(* IEC 61131-3 sources: ml2plc/benchmarks/st, 42 files *)

(* ---- CNN1.st ---- *)
FUNCTION_BLOCK CNN1_FB

    (* Model Inputs/Outputs *)
VAR_INPUT
    input_data : REAL;
END_VAR

VAR_OUTPUT
    output_data : ARRAY[0..2] OF REAL;
END_VAR

VAR CONSTANT
    weights_0 : ARRAY[0..5] OF REAL := [-0.757294893, 1.60322511, -0.810065687, -0.0401188135, -0.0341094136, 2.28848505];
    bias_0 : ARRAY[0..5] OF REAL := [0, -0.327996045, 0, 0, 0, -0.425784826];

    weights_2 : ARRAY[0..95] OF REAL := [0.387440026, -0.331604958, -0.485271782, -0.178175241, -0.261189312, -0.126141995, -0.41867274, 0.10701102, -0.504957795, -0.0640092492, -0.506339848, -0.0112774968, -0.248149365, 0.370121658, 0.102361083, 0.514361918, 2.27920318, -2.03401303, 2.57838869, 0.345396936, 1.7697078, 2.31489539, 1.82641065, 0.116435051, 2.60688972, -0.141314536, 0.0899649858, -0.115778536, -0.130346328, -2.0967865, 1.73134959, 1.73764074, -0.125548214, -0.418661654, 0.42383492, 0.245940804, -0.231652409, -0.521428883, -0.369046271, 0.500959337, 0.39457792, -0.498766184, 0.505615175, 0.00158774853, -0.358177781, 0.0681350231, 0.211269855, 0.317975223, 0.470600903, -0.22380206, -0.221884102, 0.369123101, -0.365577281, 0.470880032, 0.0877029896, -0.22456941, 0.125117779, 0.0604217052, 0.403043449, 0.0515841246, 0.360347748, 0.176390409, 0.499794424, 0.4554739, 0.357078254, -0.20554477, -0.338528842, -0.346329391, -0.316419125, -0.192169428, 0.340339243, -0.170743108, 0.503388941, 0.431303263, 0.182139158, 0.344671071, 0.0957750082, -0.455443144, 0.516620576, -0.12648204, 2.20542169, -1.42068136, 1.77867258, -0.279205918, 1.31937492, 2.40089417, 1.49984801, -0.381873012, 2.37344623, -0.157825798, -0.164687812, -0.438219547, -0.030656606, -0.809033334, 1.04967833, 1.52932751];
    bias_2 : ARRAY[0..15] OF REAL := [-0.00126687379, 1.46715438, -0.0669283643, 0, -0.544165969, -0.00420819549, -0.593534648, 0, -0.00139115693, 0, 0, 0, 0, 1.40235019, -0.471719682, -0.589310586];

    weights_3 : ARRAY[0..47] OF REAL := [-2.44326067, 1.56872427, 1.00637841, 2.21994734, -0.0721509904, -2.70681095, -2.57062817, 0.8563025, 1.35775805, 0.436492383, -0.214310527, 0.435115576, -0.357676566, -2.57688642, 2.20074344, -1.96935773, 1.55129766, 1.27391887, -0.475576401, -2.55197287, 1.79706705, -0.406806469, -0.373194754, 0.021515131, -1.98918331, 1.86888134, 1.35972965, 0.224319875, -0.156571329, -0.38576901, -0.264996111, -0.172905713, 0.307211518, 0.210194111, -0.266009122, -0.164967567, -0.275477469, 0.512401879, 0.539515197, 1.5903399, -0.0624566786, -2.02082109, -1.80255735, -3.25323439, 2.98463917, -0.251099586, -2.6509831, 1.72883391];
    bias_3 : ARRAY[0..2] OF REAL := [0.74891752, -0.036865145, -0.95004487];

END_VAR

VAR
    (* Merged variables from all regions *)
    buffer_0 : ARRAY[0..5] OF REAL;
    buffer_1 : ARRAY[0..15] OF REAL;

    (* Temporary computation variables *)
    i : DINT;
    j : DINT;
    t : DINT;
    sum : REAL;
    (* Computation helpers *)
    max_val : REAL;
    exp_val : REAL;
    exp_sum : REAL;
    (* Spatial loop variables *)
    oc : DINT;
    oh : DINT;
    ow : DINT;
    ic : DINT;
    kh : DINT;
    kw : DINT;
    ih : DINT;
    iw : DINT;
END_VAR

(* Forward pass execution *)

(* Region: r0 [ACYCLIC] *)
(* Acyclic Region r0 *)
(* Layer 0: Conv2D  in=1x1x1  out=6x1x1  kernel=1x1  stride=1x1  pad=(0, 0, 0, 0)  group=1 *)
FOR oc := 0 TO 5 DO
    FOR oh := 0 TO 0 DO
        FOR ow := 0 TO 0 DO
            sum := bias_0[oc];
            FOR ic := 0 TO 0 DO
                FOR kh := 0 TO 0 DO
                    FOR kw := 0 TO 0 DO
                        ih := oh * 1 - 0 + kh;
                        iw := ow * 1 - 0 + kw;
                        sum := sum + input_data * weights_0[oc * 1 + ic * 1 + kh * 1 + kw];
                    END_FOR;
                END_FOR;
            END_FOR;
            buffer_1[oc * 1 + oh * 1 + ow] := sum;
        END_FOR;
    END_FOR;
END_FOR;

(* Layer 1: Activation (RELU) *)
FOR i := 0 TO 5 DO
    buffer_0[i] := MAX(buffer_1[i], 0.0);
END_FOR;

(* Layer 2: Fused Linear + RELU *)
FOR j := 0 TO 15 DO
    sum := 0.0;
    FOR i := 0 TO 5 DO
        sum := sum + buffer_0[i] * weights_2[i * 16 + j];
    END_FOR;
buffer_1[j] := MAX(sum + bias_2[j], 0.0);
END_FOR;

(* Layer 3: Fused Linear + SOFTMAX *)
FOR j := 0 TO 2 DO
    sum := 0.0;
    FOR i := 0 TO 15 DO
        sum := sum + buffer_1[i] * weights_3[i * 3 + j];
    END_FOR;
output_data[j] := sum + bias_3[j];
END_FOR;

(* Softmax: find max *)
max_val := output_data[0];
FOR i := 1 TO 2 DO
    IF output_data[i] > max_val THEN
        max_val := output_data[i];
    END_IF;
END_FOR;

(* Softmax: compute exponentials and sum *)
exp_sum := 0.0;
FOR i := 0 TO 2 DO
    output_data[i] := EXP(output_data[i] - max_val);
    exp_sum := exp_sum + output_data[i];
END_FOR;

(* Softmax: normalize *)
FOR i := 0 TO 2 DO
    output_data[i] := output_data[i] / exp_sum;
END_FOR;

END_FUNCTION_BLOCK

(* ---- CNN1_straton.st ---- *)
FUNCTION_BLOCK CNN1_FB

    (* Model Inputs/Outputs *)
VAR_INPUT
    input_data : REAL;
END_VAR

VAR_OUTPUT
    output_data : ARRAY[0..2] OF REAL;
END_VAR

VAR
    CONSTANT weights_0 : ARRAY[0..5] OF REAL := [-0.757294893, 1.60322511, -0.810065687, -0.0401188135, -0.0341094136, 2.28848505];
    CONSTANT bias_0 : ARRAY[0..5] OF REAL := [0, -0.327996045, 0, 0, 0, -0.425784826];
    CONSTANT weights_2 : ARRAY[0..95] OF REAL := [0.387440026, -0.331604958, -0.485271782, -0.178175241, -0.261189312, -0.126141995, -0.41867274, 0.10701102, -0.504957795, -0.0640092492, -0.506339848, -0.0112774968, -0.248149365, 0.370121658, 0.102361083, 0.514361918, 2.27920318, -2.03401303, 2.57838869, 0.345396936, 1.7697078, 2.31489539, 1.82641065, 0.116435051, 2.60688972, -0.141314536, 0.0899649858, -0.115778536, -0.130346328, -2.0967865, 1.73134959, 1.73764074, -0.125548214, -0.418661654, 0.42383492, 0.245940804, -0.231652409, -0.521428883, -0.369046271, 0.500959337, 0.39457792, -0.498766184, 0.505615175, 0.00158774853, -0.358177781, 0.0681350231, 0.211269855, 0.317975223, 0.470600903, -0.22380206, -0.221884102, 0.369123101, -0.365577281, 0.470880032, 0.0877029896, -0.22456941, 0.125117779, 0.0604217052, 0.403043449, 0.0515841246, 0.360347748, 0.176390409, 0.499794424, 0.4554739, 0.357078254, -0.20554477, -0.338528842, -0.346329391, -0.316419125, -0.192169428, 0.340339243, -0.170743108, 0.503388941, 0.431303263, 0.182139158, 0.344671071, 0.0957750082, -0.455443144, 0.516620576, -0.12648204, 2.20542169, -1.42068136, 1.77867258, -0.279205918, 1.31937492, 2.40089417, 1.49984801, -0.381873012, 2.37344623, -0.157825798, -0.164687812, -0.438219547, -0.030656606, -0.809033334, 1.04967833, 1.52932751];
    CONSTANT bias_2 : ARRAY[0..15] OF REAL := [-0.00126687379, 1.46715438, -0.0669283643, 0, -0.544165969, -0.00420819549, -0.593534648, 0, -0.00139115693, 0, 0, 0, 0, 1.40235019, -0.471719682, -0.589310586];
    CONSTANT weights_3 : ARRAY[0..47] OF REAL := [-2.44326067, 1.56872427, 1.00637841, 2.21994734, -0.0721509904, -2.70681095, -2.57062817, 0.8563025, 1.35775805, 0.436492383, -0.214310527, 0.435115576, -0.357676566, -2.57688642, 2.20074344, -1.96935773, 1.55129766, 1.27391887, -0.475576401, -2.55197287, 1.79706705, -0.406806469, -0.373194754, 0.021515131, -1.98918331, 1.86888134, 1.35972965, 0.224319875, -0.156571329, -0.38576901, -0.264996111, -0.172905713, 0.307211518, 0.210194111, -0.266009122, -0.164967567, -0.275477469, 0.512401879, 0.539515197, 1.5903399, -0.0624566786, -2.02082109, -1.80255735, -3.25323439, 2.98463917, -0.251099586, -2.6509831, 1.72883391];
    CONSTANT bias_3 : ARRAY[0..2] OF REAL := [0.74891752, -0.036865145, -0.95004487];
END_VAR

VAR
    (* Merged variables from all regions *)
    buffer_0 : ARRAY[0..5] OF REAL;
    buffer_1 : ARRAY[0..15] OF REAL;

    (* Temporary computation variables *)
    i : DINT;
    j : DINT;
    t : DINT;
    sum : REAL;
    (* Computation helpers *)
    max_val : REAL;
    exp_val : REAL;
    exp_sum : REAL;
    (* Spatial loop variables *)
    oc : DINT;
    oh : DINT;
    ow : DINT;
    ic : DINT;
    kh : DINT;
    kw : DINT;
    ih : DINT;
    iw : DINT;
END_VAR

(* Forward pass execution *)

(* Region: r0 [ACYCLIC] *)
(* Acyclic Region r0 *)
(* Layer 0: Conv2D  in=1x1x1  out=6x1x1  kernel=1x1  stride=1x1  pad=(0, 0, 0, 0)  group=1 *)
FOR oc := 0 TO 5 DO
    FOR oh := 0 TO 0 DO
        FOR ow := 0 TO 0 DO
            sum := bias_0[oc];
            FOR ic := 0 TO 0 DO
                FOR kh := 0 TO 0 DO
                    FOR kw := 0 TO 0 DO
                        ih := oh * 1 - 0 + kh;
                        iw := ow * 1 - 0 + kw;
                        sum := sum + input_data * weights_0[oc * 1 + ic * 1 + kh * 1 + kw];
                    END_FOR;
                END_FOR;
            END_FOR;
            buffer_1[oc * 1 + oh * 1 + ow] := sum;
        END_FOR;
    END_FOR;
END_FOR;

(* Layer 1: Activation (RELU) *)
FOR i := 0 TO 5 DO
    buffer_0[i] := MAX(buffer_1[i], 0.0);
END_FOR;

(* Layer 2: Fused Linear + RELU *)
FOR j := 0 TO 15 DO
    sum := 0.0;
    FOR i := 0 TO 5 DO
        sum := sum + buffer_0[i] * weights_2[i * 16 + j];
    END_FOR;
buffer_1[j] := MAX(sum + bias_2[j], 0.0);
END_FOR;

(* Layer 3: Fused Linear + SOFTMAX *)
FOR j := 0 TO 2 DO
    sum := 0.0;
    FOR i := 0 TO 15 DO
        sum := sum + buffer_1[i] * weights_3[i * 3 + j];
    END_FOR;
output_data[j] := sum + bias_3[j];
END_FOR;

(* Softmax: find max *)
max_val := output_data[0];
FOR i := 1 TO 2 DO
    IF output_data[i] > max_val THEN
        max_val := output_data[i];
    END_IF;
END_FOR;

(* Softmax: compute exponentials and sum *)
exp_sum := 0.0;
FOR i := 0 TO 2 DO
    output_data[i] := EXP(output_data[i] - max_val);
    exp_sum := exp_sum + output_data[i];
END_FOR;

(* Softmax: normalize *)
FOR i := 0 TO 2 DO
    output_data[i] := output_data[i] / exp_sum;
END_FOR;

END_FUNCTION_BLOCK

(* ---- CNN2.st ---- *)
FUNCTION_BLOCK CNN2_FB

    (* Model Inputs/Outputs *)
VAR_INPUT
    input_data : REAL;
END_VAR

VAR_OUTPUT
    output_data : ARRAY[0..2] OF REAL;
END_VAR

VAR CONSTANT
    weights_0 : ARRAY[0..9] OF REAL := [-0.262705386, 0.779935002, 1.03506529, 0.632895529, -0.312737316, -0.310815006, 1.04849136, 0.870586991, -0.33241713, 0.675958574];
    bias_0 : ARRAY[0..9] OF REAL := [0, -0.171853036, 0.155731231, -0.141236976, 0, 0.388507366, -0.176535189, -0.0690641031, 0, -0.149513766];

    weights_2 : ARRAY[0..99] OF REAL := [-0.0687341988, -0.505324185, -0.171715677, -0.380084217, 0.443206012, -0.165993631, -0.00731980801, -0.294861794, -0.329322875, -0.340971529, -0.39975965, -1.21721697, 0.0680034459, -1.40909934, 0.224685371, 0.851948142, -0.889827847, -0.095493108, -0.157179385, -1.28536439, -0.545177042, -1.34768605, 0.0538454317, -0.994832158, 0.527012348, 0.700168669, -1.15851235, -0.457079113, -0.00149732828, -0.467484027, 0.178472638, -1.06804824, 0.428462833, -0.918258965, -0.139204293, 0.417420805, -0.467564315, 0.0089803664, -0.24426356, -1.38583362, -0.463089764, 0.807691395, 0.923243821, 0.796885252, 0.0120127201, -0.49810043, 0.873528719, 0.914482772, 0.53928721, 0.734467626, 0.278324604, 1.19621909, 0.403788477, 1.62108636, 0.500351071, -0.523164451, 0.972507596, 0.644115269, -0.138118327, 1.47070789, 0.209766984, 0.853332102, 0.699123144, 0.846534193, 0.213573575, 0.678547621, 1.08085775, 0.551357388, 0.0911467671, 0.56043458, 0.102282166, 0.877178192, 1.12506092, 0.902248561, 0.383322537, 0.205958784, 1.27946091, 0.450389624, 0.0967945457, 1.4164356, -0.126412362, 0.519436717, -0.367547452, -0.315561593, 0.464017153, -0.335243285, -0.132026047, 0.0108332634, -0.113086581, 0.499188185, -0.124567181, 0.982846677, 0.764017642, 0.814776838, 0.0450161695, -0.607075572, 1.12853694, 1.060583, -0.528354645, 1.37106454];
    bias_2 : ARRAY[0..9] OF REAL := [0, 0.411672026, 0.443880588, 0.573848665, -0.0798636526, -0.125108838, 0.121025026, 0.385259449, 0, -0.19617413];

    weights_4 : ARRAY[0..159] OF REAL := [-0.201477349, 0.413015246, 0.0206950307, -0.0461762249, 0.247961462, -0.0568501949, 0.0383369327, -0.259854972, -0.444527179, 0.354037642, -0.150492162, -0.45852077, -0.0717066824, 0.0723364949, -0.436497748, 0.205825031, -0.853246808, -0.203027666, 1.20550728, -0.617461145, -0.294606566, -0.758126974, -0.360774875, 1.18120348, -0.898286581, 0.0282400548, -1.29355359, -1.02225327, 1.36176789, -1.26122117, 0.888965607, 1.20138299, -0.437244713, 0.199938715, 0.952059329, -0.784977317, 0.0588901639, -1.04772234, 0.136933327, 1.38765883, -1.02401209, -0.190438345, -1.35698009, -0.895844221, 1.04432738, -1.36716759, 0.705555797, 1.05620801, -0.371350586, -0.352627158, 0.698318362, 0.339798629, 0.122619152, -0.237219259, -0.306308031, 1.1137104, -0.832840025, 0.156991944, -0.679998279, 0.0465113483, 1.23213017, -0.571536481, 0.246266142, 0.828268647, 0.954969525, -0.441162556, -0.358765662, 1.20794833, 0.110377789, 1.0829252, 0.405489266, -0.158480242, 0.666661501, 0.0484011397, 0.520474494, 1.13683498, 0.0207684785, 0.065361008, -1.06433892, -0.351153046, 0.922352195, 0.37286973, -1.06930172, 1.45499146, 0.0288344026, 0.683918893, 0.106652997, -1.36949015, 0.743930757, -0.0947244018, 1.00891256, 1.05642653, -0.428952485, 1.03859484, -1.48183143, -0.854047179, 0.968141913, -0.342124283, -0.0926529169, 0.195784971, -0.294896543, 0.739876568, 0.0116237206, 0.40778929, 0.354515821, -0.374024361, 0.515046716, 0.514852107, 0.0310237482, 0.347146124, 0.0413676128, 0.718492866, 0.93554163, -0.22991991, 0.326657355, 0.398625523, 0.118993759, 0.517512321, -0.135471746, -0.152048439, -0.0744148493, 0.283234626, -0.0480741784, 0.59221071, 0.0835574865, 0.334898084, 0.113840885, 0.6169101, -0.2696082, -0.247115731, -0.115800917, -0.455095321, 0.19553715, 0.408255994, -0.273867786, 0.301775157, 0.0945883393, -0.105913788, -0.189621061, 0.266120255, 0.308612525, 0.111635566, -0.232673854, 0.203693449, 0.932905853, 0.0795902014, -0.982003152, 1.30284607, -0.24889259, 0.664860845, -0.268993974, -1.18393588, 0.884641588, -0.373547137, 0.737916648, 0.872539937, -0.961955905, 0.336005777, -1.42044866, -0.375628591];
    bias_4 : ARRAY[0..15] OF REAL := [0.0454013124, 0, 0.330961257, 0.0879051089, 0, -0.0268695857, -0.00847197231, 0.40490979, -0.30825153, -0.0550679453, -0.272085756, 0.118456185, 0.399625003, -0.25876981, 0.0508395843, 0.437826991];

    weights_5 : ARRAY[0..47] OF REAL := [-1.41491461, 0.827757239, 0.660482943, -0.25115788, -0.280392915, 0.466725051, 1.23645818, -0.262650639, -1.58302641, -1.17853892, 0.55448246, 0.658791304, 0.462803185, 0.334367275, -0.154009759, -1.42141747, 0.455798388, 1.09709466, -0.269543529, 0.381915301, 0.213490352, 0.856128395, -0.295868725, -1.65038943, -0.223673388, -1.45374537, 0.96670717, 0.0626830533, 0.351752698, 0.458376706, -0.513772011, -1.85208988, 0.897746146, -1.27468288, 0.557765663, 0.871361613, 0.802684307, 0.374990225, -1.3816756, -0.737900555, -1.92418301, 1.15498805, 1.33344316, -2.06843209, -0.317642659, 0.74203372, 0.87400955, -0.946626067];
    bias_5 : ARRAY[0..2] OF REAL := [0.00161235163, 0.236852512, -0.336925507];

END_VAR

VAR
    (* Merged variables from all regions *)
    buffer_0 : ARRAY[0..9] OF REAL;
    buffer_1 : ARRAY[0..15] OF REAL;

    (* Temporary computation variables *)
    i : DINT;
    j : DINT;
    t : DINT;
    sum : REAL;
    (* Computation helpers *)
    max_val : REAL;
    exp_val : REAL;
    exp_sum : REAL;
    (* Spatial loop variables *)
    oc : DINT;
    oh : DINT;
    ow : DINT;
    ic : DINT;
    kh : DINT;
    kw : DINT;
    ih : DINT;
    iw : DINT;
END_VAR

(* Forward pass execution *)

(* Region: r0 [ACYCLIC] *)
(* Acyclic Region r0 *)
(* Layer 0: Conv2D  in=1x1x1  out=10x1x1  kernel=1x1  stride=1x1  pad=(0, 0, 0, 0)  group=1 *)
FOR oc := 0 TO 9 DO
    FOR oh := 0 TO 0 DO
        FOR ow := 0 TO 0 DO
            sum := bias_0[oc];
            FOR ic := 0 TO 0 DO
                FOR kh := 0 TO 0 DO
                    FOR kw := 0 TO 0 DO
                        ih := oh * 1 - 0 + kh;
                        iw := ow * 1 - 0 + kw;
                        sum := sum + input_data * weights_0[oc * 1 + ic * 1 + kh * 1 + kw];
                    END_FOR;
                END_FOR;
            END_FOR;
            buffer_1[oc * 1 + oh * 1 + ow] := sum;
        END_FOR;
    END_FOR;
END_FOR;

(* Layer 1: Activation (RELU) *)
FOR i := 0 TO 9 DO
    buffer_0[i] := MAX(buffer_1[i], 0.0);
END_FOR;

(* Layer 2: Conv2D  in=10x1x1  out=10x1x1  kernel=1x1  stride=1x1  pad=(0, 0, 0, 0)  group=1 *)
FOR oc := 0 TO 9 DO
    FOR oh := 0 TO 0 DO
        FOR ow := 0 TO 0 DO
            sum := bias_2[oc];
            FOR ic := 0 TO 9 DO
                FOR kh := 0 TO 0 DO
                    FOR kw := 0 TO 0 DO
                        ih := oh * 1 - 0 + kh;
                        iw := ow * 1 - 0 + kw;
                        sum := sum + buffer_0[ic * 1 + ih * 1 + iw] * weights_2[oc * 10 + ic * 1 + kh * 1 + kw];
                    END_FOR;
                END_FOR;
            END_FOR;
            buffer_1[oc * 1 + oh * 1 + ow] := sum;
        END_FOR;
    END_FOR;
END_FOR;

(* Layer 3: Activation (RELU) *)
FOR i := 0 TO 9 DO
    buffer_0[i] := MAX(buffer_1[i], 0.0);
END_FOR;

(* Layer 4: Fused Linear + RELU *)
FOR j := 0 TO 15 DO
    sum := 0.0;
    FOR i := 0 TO 9 DO
        sum := sum + buffer_0[i] * weights_4[i * 16 + j];
    END_FOR;
buffer_1[j] := MAX(sum + bias_4[j], 0.0);
END_FOR;

(* Layer 5: Fused Linear + SOFTMAX *)
FOR j := 0 TO 2 DO
    sum := 0.0;
    FOR i := 0 TO 15 DO
        sum := sum + buffer_1[i] * weights_5[i * 3 + j];
    END_FOR;
output_data[j] := sum + bias_5[j];
END_FOR;

(* Softmax: find max *)
max_val := output_data[0];
FOR i := 1 TO 2 DO
    IF output_data[i] > max_val THEN
        max_val := output_data[i];
    END_IF;
END_FOR;

(* Softmax: compute exponentials and sum *)
exp_sum := 0.0;
FOR i := 0 TO 2 DO
    output_data[i] := EXP(output_data[i] - max_val);
    exp_sum := exp_sum + output_data[i];
END_FOR;

(* Softmax: normalize *)
FOR i := 0 TO 2 DO
    output_data[i] := output_data[i] / exp_sum;
END_FOR;

END_FUNCTION_BLOCK

(* ---- CNN2_straton.st ---- *)
FUNCTION_BLOCK CNN2_FB

    (* Model Inputs/Outputs *)
VAR_INPUT
    input_data : REAL;
END_VAR

VAR_OUTPUT
    output_data : ARRAY[0..2] OF REAL;
END_VAR

VAR
    CONSTANT weights_0 : ARRAY[0..9] OF REAL := [-0.262705386, 0.779935002, 1.03506529, 0.632895529, -0.312737316, -0.310815006, 1.04849136, 0.870586991, -0.33241713, 0.675958574];
    CONSTANT bias_0 : ARRAY[0..9] OF REAL := [0, -0.171853036, 0.155731231, -0.141236976, 0, 0.388507366, -0.176535189, -0.0690641031, 0, -0.149513766];
    CONSTANT weights_2 : ARRAY[0..99] OF REAL := [-0.0687341988, -0.505324185, -0.171715677, -0.380084217, 0.443206012, -0.165993631, -0.00731980801, -0.294861794, -0.329322875, -0.340971529, -0.39975965, -1.21721697, 0.0680034459, -1.40909934, 0.224685371, 0.851948142, -0.889827847, -0.095493108, -0.157179385, -1.28536439, -0.545177042, -1.34768605, 0.0538454317, -0.994832158, 0.527012348, 0.700168669, -1.15851235, -0.457079113, -0.00149732828, -0.467484027, 0.178472638, -1.06804824, 0.428462833, -0.918258965, -0.139204293, 0.417420805, -0.467564315, 0.0089803664, -0.24426356, -1.38583362, -0.463089764, 0.807691395, 0.923243821, 0.796885252, 0.0120127201, -0.49810043, 0.873528719, 0.914482772, 0.53928721, 0.734467626, 0.278324604, 1.19621909, 0.403788477, 1.62108636, 0.500351071, -0.523164451, 0.972507596, 0.644115269, -0.138118327, 1.47070789, 0.209766984, 0.853332102, 0.699123144, 0.846534193, 0.213573575, 0.678547621, 1.08085775, 0.551357388, 0.0911467671, 0.56043458, 0.102282166, 0.877178192, 1.12506092, 0.902248561, 0.383322537, 0.205958784, 1.27946091, 0.450389624, 0.0967945457, 1.4164356, -0.126412362, 0.519436717, -0.367547452, -0.315561593, 0.464017153, -0.335243285, -0.132026047, 0.0108332634, -0.113086581, 0.499188185, -0.124567181, 0.982846677, 0.764017642, 0.814776838, 0.0450161695, -0.607075572, 1.12853694, 1.060583, -0.528354645, 1.37106454];
    CONSTANT bias_2 : ARRAY[0..9] OF REAL := [0, 0.411672026, 0.443880588, 0.573848665, -0.0798636526, -0.125108838, 0.121025026, 0.385259449, 0, -0.19617413];
    CONSTANT weights_4 : ARRAY[0..159] OF REAL := [-0.201477349, 0.413015246, 0.0206950307, -0.0461762249, 0.247961462, -0.0568501949, 0.0383369327, -0.259854972, -0.444527179, 0.354037642, -0.150492162, -0.45852077, -0.0717066824, 0.0723364949, -0.436497748, 0.205825031, -0.853246808, -0.203027666, 1.20550728, -0.617461145, -0.294606566, -0.758126974, -0.360774875, 1.18120348, -0.898286581, 0.0282400548, -1.29355359, -1.02225327, 1.36176789, -1.26122117, 0.888965607, 1.20138299, -0.437244713, 0.199938715, 0.952059329, -0.784977317, 0.0588901639, -1.04772234, 0.136933327, 1.38765883, -1.02401209, -0.190438345, -1.35698009, -0.895844221, 1.04432738, -1.36716759, 0.705555797, 1.05620801, -0.371350586, -0.352627158, 0.698318362, 0.339798629, 0.122619152, -0.237219259, -0.306308031, 1.1137104, -0.832840025, 0.156991944, -0.679998279, 0.0465113483, 1.23213017, -0.571536481, 0.246266142, 0.828268647, 0.954969525, -0.441162556, -0.358765662, 1.20794833, 0.110377789, 1.0829252, 0.405489266, -0.158480242, 0.666661501, 0.0484011397, 0.520474494, 1.13683498, 0.0207684785, 0.065361008, -1.06433892, -0.351153046, 0.922352195, 0.37286973, -1.06930172, 1.45499146, 0.0288344026, 0.683918893, 0.106652997, -1.36949015, 0.743930757, -0.0947244018, 1.00891256, 1.05642653, -0.428952485, 1.03859484, -1.48183143, -0.854047179, 0.968141913, -0.342124283, -0.0926529169, 0.195784971, -0.294896543, 0.739876568, 0.0116237206, 0.40778929, 0.354515821, -0.374024361, 0.515046716, 0.514852107, 0.0310237482, 0.347146124, 0.0413676128, 0.718492866, 0.93554163, -0.22991991, 0.326657355, 0.398625523, 0.118993759, 0.517512321, -0.135471746, -0.152048439, -0.0744148493, 0.283234626, -0.0480741784, 0.59221071, 0.0835574865, 0.334898084, 0.113840885, 0.6169101, -0.2696082, -0.247115731, -0.115800917, -0.455095321, 0.19553715, 0.408255994, -0.273867786, 0.301775157, 0.0945883393, -0.105913788, -0.189621061, 0.266120255, 0.308612525, 0.111635566, -0.232673854, 0.203693449, 0.932905853, 0.0795902014, -0.982003152, 1.30284607, -0.24889259, 0.664860845, -0.268993974, -1.18393588, 0.884641588, -0.373547137, 0.737916648, 0.872539937, -0.961955905, 0.336005777, -1.42044866, -0.375628591];
    CONSTANT bias_4 : ARRAY[0..15] OF REAL := [0.0454013124, 0, 0.330961257, 0.0879051089, 0, -0.0268695857, -0.00847197231, 0.40490979, -0.30825153, -0.0550679453, -0.272085756, 0.118456185, 0.399625003, -0.25876981, 0.0508395843, 0.437826991];
    CONSTANT weights_5 : ARRAY[0..47] OF REAL := [-1.41491461, 0.827757239, 0.660482943, -0.25115788, -0.280392915, 0.466725051, 1.23645818, -0.262650639, -1.58302641, -1.17853892, 0.55448246, 0.658791304, 0.462803185, 0.334367275, -0.154009759, -1.42141747, 0.455798388, 1.09709466, -0.269543529, 0.381915301, 0.213490352, 0.856128395, -0.295868725, -1.65038943, -0.223673388, -1.45374537, 0.96670717, 0.0626830533, 0.351752698, 0.458376706, -0.513772011, -1.85208988, 0.897746146, -1.27468288, 0.557765663, 0.871361613, 0.802684307, 0.374990225, -1.3816756, -0.737900555, -1.92418301, 1.15498805, 1.33344316, -2.06843209, -0.317642659, 0.74203372, 0.87400955, -0.946626067];
    CONSTANT bias_5 : ARRAY[0..2] OF REAL := [0.00161235163, 0.236852512, -0.336925507];
END_VAR

VAR
    (* Merged variables from all regions *)
    buffer_0 : ARRAY[0..9] OF REAL;
    buffer_1 : ARRAY[0..15] OF REAL;

    (* Temporary computation variables *)
    i : DINT;
    j : DINT;
    t : DINT;
    sum : REAL;
    (* Computation helpers *)
    max_val : REAL;
    exp_val : REAL;
    exp_sum : REAL;
    (* Spatial loop variables *)
    oc : DINT;
    oh : DINT;
    ow : DINT;
    ic : DINT;
    kh : DINT;
    kw : DINT;
    ih : DINT;
    iw : DINT;
END_VAR

(* Forward pass execution *)

(* Region: r0 [ACYCLIC] *)
(* Acyclic Region r0 *)
(* Layer 0: Conv2D  in=1x1x1  out=10x1x1  kernel=1x1  stride=1x1  pad=(0, 0, 0, 0)  group=1 *)
FOR oc := 0 TO 9 DO
    FOR oh := 0 TO 0 DO
        FOR ow := 0 TO 0 DO
            sum := bias_0[oc];
            FOR ic := 0 TO 0 DO
                FOR kh := 0 TO 0 DO
                    FOR kw := 0 TO 0 DO
                        ih := oh * 1 - 0 + kh;
                        iw := ow * 1 - 0 + kw;
                        sum := sum + input_data * weights_0[oc * 1 + ic * 1 + kh * 1 + kw];
                    END_FOR;
                END_FOR;
            END_FOR;
            buffer_1[oc * 1 + oh * 1 + ow] := sum;
        END_FOR;
    END_FOR;
END_FOR;

(* Layer 1: Activation (RELU) *)
FOR i := 0 TO 9 DO
    buffer_0[i] := MAX(buffer_1[i], 0.0);
END_FOR;

(* Layer 2: Conv2D  in=10x1x1  out=10x1x1  kernel=1x1  stride=1x1  pad=(0, 0, 0, 0)  group=1 *)
FOR oc := 0 TO 9 DO
    FOR oh := 0 TO 0 DO
        FOR ow := 0 TO 0 DO
            sum := bias_2[oc];
            FOR ic := 0 TO 9 DO
                FOR kh := 0 TO 0 DO
                    FOR kw := 0 TO 0 DO
                        ih := oh * 1 - 0 + kh;
                        iw := ow * 1 - 0 + kw;
                        sum := sum + buffer_0[ic * 1 + ih * 1 + iw] * weights_2[oc * 10 + ic * 1 + kh * 1 + kw];
                    END_FOR;
                END_FOR;
            END_FOR;
            buffer_1[oc * 1 + oh * 1 + ow] := sum;
        END_FOR;
    END_FOR;
END_FOR;

(* Layer 3: Activation (RELU) *)
FOR i := 0 TO 9 DO
    buffer_0[i] := MAX(buffer_1[i], 0.0);
END_FOR;

(* Layer 4: Fused Linear + RELU *)
FOR j := 0 TO 15 DO
    sum := 0.0;
    FOR i := 0 TO 9 DO
        sum := sum + buffer_0[i] * weights_4[i * 16 + j];
    END_FOR;
buffer_1[j] := MAX(sum + bias_4[j], 0.0);
END_FOR;

(* Layer 5: Fused Linear + SOFTMAX *)
FOR j := 0 TO 2 DO
    sum := 0.0;
    FOR i := 0 TO 15 DO
        sum := sum + buffer_1[i] * weights_5[i * 3 + j];
    END_FOR;
output_data[j] := sum + bias_5[j];
END_FOR;

(* Softmax: find max *)
max_val := output_data[0];
FOR i := 1 TO 2 DO
    IF output_data[i] > max_val THEN
        max_val := output_data[i];
    END_IF;
END_FOR;

(* Softmax: compute exponentials and sum *)
exp_sum := 0.0;
FOR i := 0 TO 2 DO
    output_data[i] := EXP(output_data[i] - max_val);
    exp_sum := exp_sum + output_data[i];
END_FOR;

(* Softmax: normalize *)
FOR i := 0 TO 2 DO
    output_data[i] := output_data[i] / exp_sum;
END_FOR;

END_FUNCTION_BLOCK

(* ---- CNN3.st ---- *)
FUNCTION_BLOCK CNN3_FB

    (* Model Inputs/Outputs *)
VAR_INPUT
    input_data : REAL;
END_VAR

VAR_OUTPUT
    output_data : ARRAY[0..2] OF REAL;
END_VAR

VAR CONSTANT
    weights_0 : ARRAY[0..31] OF REAL := [-0.305521011, -0.422613502, -0.232975915, -0.320694596, 0.165935397, -0.269291103, 0.566170037, -0.400613427, 0.189311981, -0.0100060701, -0.173879772, -0.164011866, 0.62322247, -0.0581877828, -0.14924413, 0.404986084, -0.215965614, 0.317790955, -0.291711658, 0.274873227, 0.475638539, 0.492071569, 0.634018719, -0.0343125463, -0.271868944, 0.32324031, -0.300987601, 0.309288561, -0.408682555, 0.32534194, 0.1631006, 0.26265505];
    bias_0 : ARRAY[0..31] OF REAL := [0, 0, 0, 0, 0.172577351, 0, -0.0827501416, 0, 0.223048955, 0, 0, 0, -0.105154268, 0, 0, -0.0659836903, 0, -0.0452738144, 0, -0.0564793386, -0.00329497736, -0.0965443105, -0.0831072181, 0, 0, -0.0714189336, 0, -0.0674561262, 0, -0.0654055476, 0.227993011, -0.0599486753];

    weights_2 : ARRAY[0..1023] OF REAL := [-0.302535117, 0.18892476, 0.0559765399, -0.00583121181, -0.209280849, 0.197514027, -0.0585472584, 0.226948529, -0.0109393299, -0.0708717257, -0.000990241766, -0.199344471, -0.204100311, -0.24769415, 0.196327895, 0.0838947892, -0.161202446, -0.168231815, -0.227868319, 0.122277558, 0.0647429526, -0.28689447, -0.28050983, 0.233420163, -0.0741003156, -0.134897009, -0.104453847, -0.114217952, 0.163484365, -0.12216346, 0.0639127195, 0.145405054, -0.290665954, 0.143932939, -0.0299953222, 0.235896617, -0.282639861, -0.148633957, 0.0376873016, 0.156656623, -0.0985182375, -0.0435509086, -0.015540868, 0.190203637, -0.192348331, -0.286105692, 0.273440748, -0.305073559, 0.264027983, -0.2744914, -0.254760683, -0.0749585778, -0.0793877393, -0.0355826914, 0.193246961, -0.0812891126, 0.0125352144, -0.220631987, -0.185660452, -0.0836507529, -0.287493646, 0.0952782035, 0.120691627, -0.260108113, 0.179627776, 0.0708105564, -0.218895897, 0.278866738, 0.276239067, -0.133862078, 0.0681913495, 0.00870683789, -0.268055528, -0.279873997, 0.231311589, -0.231229186, 0.103336632, -0.237921149, -0.255749762, -0.166464254, -0.163067028, 0.131616294, -0.145967394, -0.187863171, 0.20904544, -0.296933353, -0.301976651, 0.274004668, -0.0851544887, 0.303235918, -0.26501739, -0.0701736808, -0.257095665, 0.151182264, -0.157260641, 0.149946868, 0.249261647, -0.296775579, -0.111859664, -0.043521136, -0.0558283627, 0.243011326, -0.117863595, 0.137829065, -0.0363067091, 0.209354728, 0.262005001, -0.0820820332, -0.199815333, -0.298343062, -0.196902096, 0.163581759, -0.244165748, -0.208579481, 0.0648718774, 0.0387138426, 0.0587200522, 0.199852854, -0.200009495, 0.264581591, 0.157567024, -0.140247881, 0.136465728, -0.291744113, 0.199463874, -0.17022939, -0.209436268, 0.0697534382, 0.287504464, -0.239274785, 0.0915648043, -0.272040695, -0.147038579, -0.119065329, -0.453846484, -0.0374956727, 0.137012199, -0.212714791, -0.267802566, -0.286457181, -0.22830689, -0.00203335285, -0.110627413, -0.280225068, -0.0671572387, -0.375999659, -0.287249386, -0.515549958, -0.157999471, -0.441203892, 0.0731154978, 0.27118066, -0.183265448, -0.545777202, -0.284385741, -0.555042386, 0.0339722335, -0.39134109, 0.316408813, -0.51222688, 0.136596113, -0.212152988, -0.299960375, -0.126898065, 0.116992414, 0.0458351076, -0.0269443989, -0.065452233, -0.281665444, 0.0354217291, 0.18740195, 0.1303747, -0.27631107, 0.299713761, -0.190243363, 0.00589945912, -0.0832127482, -0.17362465, -0.285472333, 0.29846403, -0.247270525, 0.150024831, 0.211201519, 0.275536805, -0.264383584, 0.195956439, -0.2281674, -0.103786692, 0.290275723, -0.0386345685, 0.0585829616, -0.0255514085, 0.162740201, 0.292739421, 0.189756721, 0.252827317, 0.234207675, -0.257683247, 0.273965418, 0.0257166922, -0.036956422, 0.108332217, 0.282296747, 0.27142027, 0.179358244, 0.190752685, 0.130160302, 0.657829762, 0.214174837, 0.299848855, -0.0442554355, 0.389891922, 0.502143204, 0.627101123, 0.617687285, 0.103749901, -0.0610816926, 0.526211083, -0.119288921, 0.190606341, -0.156062484, 0.553908527, 0.227522269, 0.609408021, -0.166023687, 0.0483898222, -0.169464931, -0.202580005, 0.116183177, -0.14569962, 0.387277544, -0.155328169, 0.409152329, -0.200958371, 0.0662257373, 0.00956270099, 0.0667660981, 0.050966531, 0.252343684, 0.0681977794, 0.0483501852, 0.467907012, -0.192403793, 0.353288114, 0.321424454, -0.0361318104, 0.237703666, -0.0217028856, -0.179048359, -0.182526037, -0.00862252712, 0.0644219592, 0.0776462257, -0.0794326067, 0.387354374, -0.172654673, 0.166961968, -0.0229187906, -0.278536558, 0.202470273, -0.242246509, 0.00352868438, 0.0825264975, -0.169674367, -0.0711229518, 0.0518683195, -0.110450983, 0.196748346, 0.115502901, 0.0190000534, -0.272912979, 0.0419930816, 0.254024237, -0.159889773, 0.265684694, -0.0409128964, -0.29967609, 0.00678181648, -0.223878056, -0.0868313015, 0.17442584, -0.0355110168, 0.0499511063, -0.0420474112, -0.00389733911, -0.283686012, 0.274984717, -0.158691674, 0.273474425, -0.235847771, -0.250777483, -0.0218633413, 0.0308788847, -0.302752227, -0.205767021, -0.0621758997, 0.339249223, 0.239462107, -0.244065732, 0.206250519, -0.0809870958, 0.0378507376, 0.259526581, -0.350233167, -0.10086973, -0.190593183, -0.196929902, -0.364800125, -0.327376693, -0.460740179, -0.348780066, -0.304304481, -0.275294036, -0.419785649, -0.0145461559, -0.0663260296, 0.253250867, -0.235067278, -0.215728268, -0.225787237, -0.00937449932, -0.180815846, 0.0139636099, 0.17749083, 0.0060210824, -0.223020792, 0.151658207, -0.0924022645, -0.0592324436, 0.103573889, -0.0989728123, -0.166958094, -0.162929133, -0.299686998, -0.172253996, 0.201589018, -0.174295232, -0.198272675, 0.27946493, 0.113219529, -0.243771985, -0.163556278, -0.0839572698, 0.00705915689, 0.0495300293, 0.140405416, 0.196302861, 0.160213143, -0.289103985, 0.0973640382, -0.0314720571, -0.138745815, -0.263403207, -0.286320388, 0.179950446, 0.259577304, 0.221186474, 0.279502958, 0.402291119, -0.174203902, 0.367326111, 0.162910938, -0.113503411, -0.0146658719, 0.10874512, 0.0420466065, -0.224053681, 0.182572201, 0.0115836561, 0.471963674, 0.254551619, 0.642762184, 0.122648776, 0.524187386, 0.477656454, 0.281031221, -0.19247067, 0.346408755, -0.217598528, 0.355205953, -0.239685863, 0.437059462, 0.121007852, 0.481753826, 0.059666872, -0.28007251, 0.26986894, -0.29868719, 0.251580834, -0.126799658, 0.184885204, -0.283049762, 0.217957839, 0.205171674, 0.189562619, 0.036806047, 0.542116702, 0.245351404, 0.00321984291, 0.110237487, -0.243030667, 0.381333739, 0.0344565213, 0.650871336, 0.483460665, 0.586772025, 0.218027562, 0.262780279, -0.294995397, 0.376155823, 0.242882341, 0.60048157, -0.230364054, 0.561005712, -0.180027649, 0.328136921, 0.29206273, -0.0110495687, 0.185954124, -0.289577752, -0.0824203864, -0.218502581, 0.491475344, -0.239469185, -0.14291954, -0.042076081, -0.229130924, -0.0268279612, 0.456320733, 0.0788233578, -0.193412885, 0.192516625, -0.116849899, 0.357412398, 0.18516925, 0.664660394, 0.47820729, 0.219199926, 0.569181979, -0.24115178, 0.000183165073, 0.527471364, 0.217652768, 0.637461603, -0.0239106417, 0.333134413, -0.012003256, 0.762007594, -0.305104792, -0.134593263, -0.0691054016, -0.182842419, 0.104011118, -0.114199772, -0.144061953, 0.0103146136, 0.0743029416, -0.073059395, -0.302777171, -0.148231506, -0.581851542, 0.0359168351, -0.0594537854, -0.311178058, 0.115716219, -0.229913637, -0.124246091, -0.588294506, -0.144168273, -0.288753003, -0.298907161, 0.288104385, 0.188650638, -0.191782191, -0.0437152386, -0.543406188, 0.0419805348, -0.470147073, 0.231057882, -0.51450932, 0.17264542, -0.175306141, 0.173843056, 0.0492859781, 0.23577337, 0.267599136, -0.477695316, -0.230120152, 0.217158318, -0.271804094, 0.0695960224, -0.0244961083, -0.506193578, 0.135770679, 0.0872241259, -0.566133738, -0.201745093, -0.135925472, 0.0788646042, -0.539860368, -0.105563179, -0.606840909, -0.387925804, 0.0368691087, -0.178178787, -0.234305128, -0.1725941, -0.0879689828, -0.204702631, -0.464641184, 0.264212668, -0.726549506, 0.220489591, -0.258909285, 0.247580558, -0.295292139, 0.0746903941, 0.276553065, -0.34599939, 0.0651829243, -0.0950947627, 0.179230362, 0.138010263, 0.207658917, -0.485984504, 0.24705717, 0.183054984, 0.0181562435, 0.023029089, -0.154695943, 0.028001368, -0.217172459, 0.108330622, -0.606546998, -0.509887576, -0.0501905382, -0.0502379835, -0.187235802, -0.0215578377, -0.205275148, 0.159722716, -0.523856878, 0.367217451, -0.374988735, -0.258188039, 0.0893038213, 0.189385593, -0.212752685, 0.222774431, -0.192041069, -0.224466607, 0.260421485, 0.0654474869, 0.201206833, -0.0600627512, 0.0909488201, -0.366285771, 0.045057863, -0.0323132873, -0.0753270537, 0.201040119, -0.37792787, -0.29401654, -0.334450126, 0.112285152, -0.495266557, -0.345330864, 0.183888078, -0.265022576, -0.5475775, -0.274378836, -0.315385282, 0.255632907, -0.578590631, 0.266971111, -0.647537172, -0.0671942532, 0.270085663, -0.248822376, 0.211921662, 0.181917012, 0.113762349, 0.254813403, -0.0133170485, -0.117874727, -0.086210072, 0.0855523348, -0.144555777, -0.0541543961, -0.289933681, 0.203286916, 0.112982489, -0.239740968, -0.174730241, 0.132769346, -0.335220218, -0.0906959474, -0.242582321, 0.216031134, 0.166696459, -0.0664575249, -0.119935647, 0.126910329, 0.166350543, -0.116871879, -0.012888276, -0.0793427974, 0.117575742, -0.160697132, 0.282213181, -0.296972394, 0.182963759, 0.136175245, 0.0425625741, 0.0446024835, 0.303385705, -0.240173712, -0.0353201032, -0.0117941797, -0.0658513308, -0.190131158, -0.0233257711, 0.0762789249, 0.130448371, 0.149402589, -0.12086077, 0.228611737, 0.0254626572, -0.142554909, 0.0261900127, 0.277120203, -0.209043026, 0.149235845, 0.0761509538, 0.0277103186, -0.0605103225, -0.017962575, -0.0947141945, -0.251718462, 0.0736608505, -0.00390675664, 0.122442633, 0.241143972, -0.0663959831, 0.275990337, -0.0487243831, 0.0234669391, -0.208523691, -0.238098904, 0.119020581, -0.292945325, -0.0633578449, -0.266576141, -0.203903496, 0.255696267, 0.247468084, 0.0727858543, 0.171153888, -0.223049626, 0.00358453393, -0.287472397, 0.16379863, -0.154578328, -0.17688185, -0.261389345, -0.199313164, -0.189400047, -0.30364421, -0.0939725786, -0.22107321, 0.0905611366, -0.00646039844, 0.284296423, -0.0867350101, 0.306169897, -0.298862249, -0.0602645464, 0.0698877573, -0.0183352437, -0.244261891, 0.286652148, -0.0848819762, 0.281890005, -0.244641051, -0.371583819, 0.0368148088, 0.111535549, -0.145513758, 0.141247839, -0.124237344, -0.199639976, -0.283237904, -0.172199294, -0.315320283, -0.465632647, 0.268095762, 0.260501713, -0.166749552, 0.0841402113, -0.323706269, 0.156345278, -0.105805621, 0.122712575, -0.238665223, 0.0484748781, 0.24705562, 0.165319085, 0.263771862, -0.174353406, -0.0772219598, -0.0862069279, -0.139451876, -0.041061312, -0.247308925, 0.133348018, -0.198757261, 0.277923077, -0.201209709, -0.180844694, -0.0163782537, 0.212465972, 0.291234404, -0.224223465, 0.245595306, -0.23642908, -0.000798106194, -0.28197524, 0.265623778, -0.14943251, -0.213474885, -0.0476028025, -0.218912333, -0.290392488, -0.0336225033, -0.226791486, -0.200182006, 0.264308125, 0.298065335, 0.160595387, -0.274919182, -0.0111782206, 0.08963269, 0.206110343, 0.232178122, 0.351918876, 0.251157731, 0.229518324, -0.162958845, 0.570871413, -0.114465863, -0.300647527, 0.387923539, -0.194804057, 0.487311661, 0.142618626, 0.296298683, 0.078456305, 0.433804035, 0.463133007, 0.0812964141, 0.297859281, 0.32541278, 0.0865969658, 0.330952734, 0.295674652, 0.28056547, -0.0745210126, 0.312628001, -0.25166291, -0.0636421144, 0.228714734, -0.0134817958, 0.446463346, -0.154749498, -0.0339341946, -0.220513672, 0.491205633, -0.034077853, -0.0826377869, 0.17509678, 0.110165067, 0.0771617293, 0.112737119, 0.0976967886, -0.101007998, 0.157721326, 0.11813283, -0.256341755, 0.0984092653, -0.249004111, -0.0396182761, 0.261826783, 0.0837214887, 0.16945079, -0.0745182335, 0.0434880741, 0.0109292567, 0.306479901, 0.456819355, -0.265923291, 0.266676933, -0.138841599, -0.231428549, 0.236799628, -0.319883972, 0.230660051, 0.113709949, 0.138469875, 0.0259396229, 0.113863736, 0.0650948882, 0.0834022462, 0.177783772, -0.209166974, 0.237130374, -0.0973150656, -0.150207549, 0.198629916, -0.00753036141, -0.326563656, 0.2125144, 0.129190043, -0.15817976, 0.22902438, -0.0657542348, -0.270366699, 0.124856383, -0.0920476913, 0.200559288, 0.272772551, -0.132015318, -0.260349125, 0.0628000498, 0.11580506, -0.155256853, -0.156667948, 0.00843694806, -0.0092907846, 0.0673252046, -0.177510321, -0.262808383, 0.216747373, 0.10598284, 0.243002325, -0.104387343, -0.0171529949, -0.157169163, 0.137609422, 0.124170989, 0.30237636, -0.186035827, 0.222451955, -0.0245195627, 0.201522022, -0.248001918, -0.0579287261, 0.175366014, -0.0383019745, 0.0974334478, -0.208626121, -0.0566462576, -0.206415594, -0.19229956, -0.0296979845, -0.118947357, -0.274238437, -0.164330587, -0.299601883, -0.103978336, -0.300699234, 0.24387376, 0.153795511, -0.0419691615, 0.263343424, 0.301897734, 0.083095789, 0.0574685931, 0.0765495598, 0.0496957302, 0.152801052, 0.126136065, -0.103010729, -0.0943269879, 0.214095294, -0.191258416, 0.267293394, -0.202065408, 0.00826314092, 0.27855882, -0.0598310493, -0.28701359, -0.239138722, -0.24846372, 0.230648041, -0.130428508, -0.0169515703, -0.0943224728, 0.303795487, 0.00882649422, 0.206780881, 0.180572346, 0.301215917, 0.0507665612, -0.0710421056, -0.0413283072, 0.242511719, 0.0594761372, -0.279334962, 0.49852708, 0.0137877464, -0.107751489, 0.49116236, 0.21107617, 0.328740776, 0.245125979, 0.676736832, 0.126276165, 0.641107976, 0.578572869, 0.0991042852, 0.117582381, 0.63090378, -0.0380260348, 0.557288527, -0.226017177, 0.296050072, 0.0576335639, 0.378168792, 0.216828078, -0.174352676, -0.122764841, 0.039359659, -0.00253027678, -0.0913577676, -0.132508948, 0.254950672, -0.286310256, -0.281505942, 0.297859162, 0.275912434, -0.272020847, -0.0592712164, 0.180334479, -0.237974942, 0.0402613878, -0.130927399, 0.197041601, 0.00459697843, 0.273145765, -0.132424995, -0.102154985, -0.0700460076, 0.291274399, 0.226469189, 0.00320282578, -0.232316315, 0.247298568, -0.152302295, -0.157789961, -0.000105053186, 0.114470959, -0.14560692, 0.105663389, -0.275510401, -0.0774826407, 0.227077276, 0.377452165, 0.198470443, 0.0355138369, 0.239741892, -0.0348302722, -0.0190246701, 0.515636384, -0.138521492, 0.0961776972, 0.324003935, 0.255324692, 0.440673292, 0.0240756273, 0.459442168, 0.282640427, 0.407175452, 0.264614642, 0.10761264, -0.247623056, 0.286343396, 0.121356964, 0.56822896, 0.147451937, 0.0539626516, 0.0242844839, 0.639796853, 0.0188569725, 0.0460903049, -0.0909120291, 0.227639169, 0.0159894601, -0.031009227, -0.436098576, 0.0352782011, 0.00297267828, -0.225614354, 0.0644460618, -0.213681251, -0.228012845, -0.251324624, -0.177940369, -0.16245681, 0.0723305643, -0.365570009, 0.13450864, -0.467065632, -0.123924538, -0.32537955, -0.0098186601, -0.0907044858, 0.0347717404, -0.593057096, 0.011321485, -0.643386543, -0.184858918, -0.227106094, 0.26758191, -0.601321578];
    bias_2 : ARRAY[0..31] OF REAL := [0, 0, 0, 0, 0.182205081, 0, 0.0261279475, 0.28638342, -0.0165894795, 0.1960399, 0, -0.0387773402, 0.0101007111, -0.00284077018, 0.160987243, 0.174085006, 0.170377508, 0.179273665, -0.0429509617, 0, -0.00890477467, 0.150043651, 0, -0.0682187304, 0.286487907, -0.0130185485, 0, -0.0115588885, -0.0444285497, 0, -0.053307794, 0.189561188];

    weights_4 : ARRAY[0..1023] OF REAL := [-0.131003603, -0.297578961, -0.26310873, -0.169719413, 0.297841758, 0.182245344, -0.184331119, -0.0984101295, 0.126124412, -0.0807622671, -0.141804472, 0.0988657176, -0.194241524, -0.220572859, -0.0358275473, -0.0211852491, 0.115968704, -0.00162622333, 0.112437308, 0.23827067, 0.0689125359, -0.0484642982, 0.0291061699, -0.270906329, -0.27576977, -0.180059344, 0.126082718, 0.301041871, -0.102828562, -0.234196514, 0.222444504, 0.0768038034, 0.273094863, 0.292191774, 0.0780140758, 0.147428423, -0.0136249661, 0.0721087158, 0.255919904, -0.0881415904, 0.0544376969, 0.0423079431, -0.148325086, -0.00977936387, -0.0138234496, -0.253410518, 0.0494041741, -0.232345223, -0.275000423, -0.111543283, -0.220192522, 0.00670334697, 0.070884645, 0.206565708, 0.217198759, -0.0778912306, -0.187225521, -0.198698565, 0.132753074, 0.0586737692, -0.0806486011, 0.152624756, -0.293686718, -0.218992561, 0.225608975, 0.0536068082, 0.0716869235, 0.154277325, 0.653066814, -0.0399393737, -0.117531918, 0.569934428, -0.162936762, 0.798092246, 0.177149475, 0.0259273723, 0.0173395667, -0.307323366, 0.565667093, 0.718658209, 0.721212089, 0.331154883, -0.113916174, 0.26572898, -0.268876523, 0.487004012, -0.108559892, -0.100212127, 0.42503354, -0.180491015, -0.184124529, -0.17368412, -0.0432037152, 0.215240985, -0.306913316, 0.640384555, -0.0745161921, 0.188456595, -0.213749588, -0.0977177173, 0.199909747, 0.2737073, -0.431319535, 0.0485795811, -0.100334682, 0.232757196, 0.00478008389, -0.228160441, -0.0320379026, -0.575055242, 0.578775227, -0.0222077891, 0.313824385, 0.275038272, 0.00503800018, -0.14406763, -0.167297617, -0.118154265, 0.0616946816, -0.429405093, 0.249885589, 0.170595288, 0.182640135, -0.0396085307, -0.512126684, 0.129387736, -0.177653104, 0.0936199725, -0.127106041, -0.297287971, -0.234297693, -0.084120065, 0.116697863, 0.025921315, -0.185892269, 0.181671292, 0.00360167027, 0.32814905, 0.223120064, -0.288998693, -0.00874315482, -0.270339459, 0.708790779, 0.161906198, 0.111572914, 0.29378131, 0.075823769, 0.140125751, -0.246390179, 0.316347033, -0.234037369, -0.253965825, 0.318873763, 0.239870697, -0.0351551473, -0.3213844, -0.460064769, -0.290605307, -0.234394252, 0.584625423, -0.242672235, -0.241201416, 0.18478474, 0.290055007, 0.163274556, 0.15410316, 0.192067057, -0.142505243, -0.192737415, -0.154993936, -0.0913852155, -0.0347047076, 0.144012079, -0.134131342, -0.25990954, -0.264261574, -0.155302331, 0.249702513, 0.11134164, -0.218827724, 0.13777405, 0.0414568782, 0.231697708, -0.076849103, 0.0426145643, 0.086880289, -0.0606261045, 0.109156653, 0.117690168, -0.260985792, -0.209287122, -0.283946246, 0.215177029, 0.0605516434, 0.0916358232, -0.133549497, 0.554910958, 0.290990323, -0.141817063, 0.0365407839, -0.045238439, 0.432281673, 0.131256342, -0.0234800465, -0.0965337977, -0.375376761, 0.525083125, 0.352996022, 0.515277684, 0.22995165, -0.0848059803, 0.0834964216, -0.0560837388, 0.131485552, 0.133105934, -0.0140744075, 0.129425555, -0.0155615378, -0.225329787, 0.270904064, -0.0891974568, 0.089304626, -0.0243603829, 0.209627539, -0.243726939, 0.189823687, 0.0152041018, -0.266784012, 0.637337625, 0.13740319, -0.207154065, 0.336286455, -0.172129199, 0.647333324, -0.170221731, 0.0529659726, 0.0119746178, -0.599500239, 0.640912414, 0.542431295, 0.25041604, 0.312373936, 0.208823249, -0.294798166, 0.132646054, 0.298118323, -0.245903745, -0.52973789, 0.332324654, 0.121275611, 0.229522377, 0.218299061, -0.401828319, 0.0384306014, -0.530368924, 0.43010512, -0.247315869, 0.124895006, 0.0318692327, 0.272524983, 0.0550513566, 0.234614164, -0.215883821, -0.244036019, -0.218965173, -0.198455393, -0.134395942, 0.151205897, 0.289359719, -0.020891428, -0.0206608176, -0.141190529, -0.119707286, -0.104627728, -0.27137807, 0.135529697, -0.0829650462, -0.0453687012, -0.04485479, -0.0753930807, -0.0144813359, -0.155932978, -0.244440377, -0.186790645, -0.210480541, 0.256311566, 0.221027821, 0.28123197, 0.280749232, 0.0854526758, 0.155673325, 0.259752721, 0.0108594894, -0.102523923, -0.127275184, -0.247410625, -0.186995566, -0.217350483, -0.0495776236, 0.0103222728, 0.266658276, -0.26752913, -0.185283333, -0.080992803, -0.158656329, 0.182905287, 0.0955551565, 0.201204032, 0.0729584992, 0.0956672728, -0.138944238, -0.112317741, -0.0252838731, -0.182611153, -0.299620211, -0.1491597, 0.122002423, 0.241469592, -0.080955714, -0.162610769, -0.146407947, 0.199809641, 0.210708469, 0.197502881, 0.838934898, 0.0320079327, -0.299073547, 0.325246692, 0.00689333631, 0.564447224, 0.197508961, 0.0743614659, 0.0179942958, -0.336701453, 0.685956359, 0.377637565, 0.7467677, 0.551242888, -0.0458685867, -0.0499052405, 0.00429141242, 0.529094696, -0.284011602, -0.164522097, 0.390723258, 0.217370152, -0.0920166671, -0.077930212, -0.0467830114, -0.216683686, -0.0916756466, 0.650523245, -0.0294721127, -0.036565721, 0.237943023, -0.107480735, 0.228550255, -0.0937533528, -0.236977115, 0.012222603, 0.0305623766, 0.0877570137, -0.177906424, -0.299257427, -0.0428002477, 0.203487545, 0.171061635, -0.0134457257, -0.307778209, 0.0998098031, -0.143109635, 0.0916756094, 0.0346160978, 0.245140105, -0.197224975, -0.13554132, -0.015408745, -0.00744786859, -0.146140918, 0.209403306, 0.05257985, 0.175278544, 0.0415592492, -0.139549226, 0.0374180079, -0.125721067, 0.128508002, -0.269290328, -0.219967037, -0.235181659, 0.250195414, -0.298137426, -0.265673667, 0.281026453, 0.248134404, 0.0835396349, 0.239232749, 0.0608434975, 0.0318036973, 0.0106616616, -0.138466731, 0.0832761824, 0.0524269044, 0.255962819, -0.201534927, 0.184504122, 0.0304804742, 0.112831086, -0.274396062, -0.138876349, 0.058968395, 0.0379446447, -0.24875623, -0.0247752666, -0.275676548, 0.0478424132, -0.175087795, 0.0343687832, 0.176422596, 0.304746062, 0.0191969275, -0.0734514892, -0.179163992, -0.175514787, -0.182104319, -0.12205182, -0.30386439, 0.247752264, -0.239594892, 0.14824459, 0.169285655, -0.229741827, -0.196575701, 0.236289904, -0.276429445, -0.176262379, 0.304197341, -0.0770847201, 0.0793125331, -0.122823998, -0.183093995, 0.288065225, -0.270255744, 0.163285434, 0.11553666, -0.064033255, -0.0639772788, 0.201865196, 0.230275959, -0.241755784, -0.241556555, 0.305846602, -0.263952911, 0.107600003, 0.428219318, 0.315932482, 0.123224176, -0.152412578, -0.194966853, -0.146775737, 0.380829424, -0.0218016729, -0.0653787628, -0.217486262, -0.208556026, 0.274650842, 0.163703889, 0.290339857, 0.274002284, -0.0617538393, 0.109624088, 0.337098092, 0.45619455, -0.291403472, 0.120722443, 0.0922868103, 0.0530038998, -0.0536386371, -0.107239835, 0.0548807606, 0.135127991, -0.00696855783, 0.305880457, 0.291272014, -0.00583931664, -0.00193941593, -0.172592193, -0.232942507, -0.282224745, 0.305994719, -0.212210357, -0.0568833984, -0.416065305, -0.260170877, 0.621187866, 0.462971807, 0.120404303, 0.219337612, -0.203068554, -0.0533760488, 0.289123356, 0.425835639, 0.251943856, -0.372243524, 0.0571667515, 0.0655154586, -0.232000068, 0.218965203, -0.587493002, 0.107556373, -0.34027192, 0.388532311, 0.0433574021, 0.0315204561, -0.175355047, -0.187859744, -0.182638451, -0.304725707, 0.570209086, 0.449475467, -0.176204562, -0.610260904, 0.0962311327, 0.106570229, 0.0998596475, 0.592721999, -0.604484499, -0.559462249, -0.528976202, -0.340306669, -0.00967260264, 0.269239873, -0.0222779214, -0.192777634, -0.265589207, 0.194036409, 0.0356762446, 0.238364995, -0.22000879, 0.187624753, 0.500942945, 0.137529343, 0.425541818, -0.384990692, 0.101938695, -0.254622191, 0.177904665, -0.301456809, 0.413415521, -0.0544238985, -0.0774152055, 0.418222398, 0.173097819, 0.517885208, -0.0749461651, -0.244810998, -0.0100581096, -0.118305884, 0.618597806, 0.39062652, 0.228008389, 0.703630686, 0.222671017, 0.0336589217, -0.209529251, 0.263971776, 0.272687167, -0.265066534, -0.0697458312, 0.245626211, -0.157372907, 0.232769161, -0.265899777, 0.212102264, -0.0321105421, 0.584425688, 0.0990063846, 0.181787193, -0.145895198, 0.212972194, 0.248728618, 0.0385749936, -0.0434899963, 0.13676697, 0.00287774205, 0.198615983, -0.0061378181, -0.24793154, 0.22239849, 0.230130091, -0.101685964, -0.154221162, 0.228392869, -0.0485958941, 0.140142381, 0.124007225, 0.186035693, -0.223669991, 0.22051391, 0.248337775, -0.255135477, 0.0779966265, -0.0259423256, 0.0840746984, -0.143623307, 0.10033232, -0.285437018, 0.0878624693, 0.112035602, -0.220232829, -0.134516388, -0.190172762, -0.441272169, -0.148970336, 0.54138267, -0.00991090573, 0.189627171, -0.407575816, 0.19614473, 0.126536384, 0.227124214, 0.299594849, -0.226639718, -0.197369441, -0.497689307, -0.170907199, -0.251754761, -0.305500329, 0.265903682, -0.258889407, 0.0551296771, 0.445930839, 0.50368911, 0.0694336891, 0.244235843, 0.169349968, 0.603258312, 0.121688455, 0.292904645, -0.432604104, -0.116104424, 0.24401471, 0.112017274, -0.0655304193, 0.0565166473, -0.159150913, 0.242028236, 0.207554147, -0.141486555, 0.183537751, 0.25860551, -0.0414259285, -0.137894377, -0.251868397, -0.252632767, 0.126727194, 0.202255249, -0.0172479134, -0.0407250747, 0.185998023, 0.241771609, -0.136747137, 0.168515861, -0.028578328, -0.282108217, -0.28433153, 0.284154743, 0.241208225, -0.283737987, -0.271706432, -0.293844461, 0.0216580406, -0.13977395, 0.119707644, 0.188743114, -0.0726560652, -0.298959702, -0.154147759, -0.0178879648, -0.207531452, 0.157043755, 0.272461146, 0.146871358, -0.144100055, -0.128470346, -0.261677355, -0.189533278, 0.0674045682, -0.125341833, -0.28721118, 0.107720211, 0.167298794, -0.140414461, 0.144382834, 0.196911126, 0.0846701041, 0.209047019, 0.226131424, 0.0532096922, 0.121982351, 0.122712441, -0.0468839705, -0.00250038318, -0.216128603, -0.0674674809, 0.0887127519, -0.103510752, -0.14008005, 0.513805509, -0.114425123, 0.404435933, 0.686877072, 0.181655616, -0.045817025, -0.0511573553, 0.577237487, 0.163091615, 0.614164174, 0.215413779, -0.000879098778, 0.290710986, 0.151218832, -0.247720852, 0.0785380006, 0.142183885, 0.495787174, -0.051781863, 0.140044674, 0.34138298, 0.0117680877, -0.167019278, 0.0618022867, 0.0912469029, -0.212469444, 0.349938422, 0.0867001414, 0.245564848, 0.182529032, 0.270203143, 0.0995755792, 0.311335832, -0.0408776402, -0.270453364, -0.0434136204, -0.0471109375, 0.39855656, -0.0565947145, 0.0709626302, -0.154750556, -0.618680537, 0.537402451, 0.495288789, 0.142095834, -0.0245976206, 0.136274114, 0.248995513, -0.228722006, 0.177052125, 0.113103449, -0.270589143, 0.0316585079, 0.0565498024, 0.168384671, -0.181288794, -0.410443008, 0.0202312171, -0.627221286, 0.341626108, -0.0968190879, 0.0112822354, 0.296315402, 0.194426328, 0.516518712, 0.0816926658, -0.371149898, -0.226421192, 0.311113507, 0.260248452, 0.135842144, -0.0135574797, -0.148965955, -0.493980706, 0.428472281, 0.442301363, 0.410756618, 0.0600324459, -0.241503343, 0.253234237, 0.191382542, 0.44889164, -0.271124542, -0.287356615, -0.0900610313, 0.222957343, -0.110820353, -0.224701554, -0.0902735591, 0.172117829, -0.0198980477, 0.0587677322, 0.261094719, 0.151453674, 0.109391958, 0.0861967206, 0.192481548, 0.0875143707, -0.186728299, -0.25434798, 0.118825734, -0.287684023, -0.271947175, -0.26722315, 0.135982662, 0.137506112, -0.239591539, -0.195562974, -0.259200782, 0.223056883, 0.151436254, 0.214638919, -0.102545604, -0.272877276, -0.00287774205, 0.194759756, -0.192125499, -0.309692442, -0.115699559, -0.0484452732, 0.118706763, 0.175819188, 0.0988839418, -0.120309293, -0.0505437851, -0.0424740314, 0.177575201, 0.114717275, -0.531936646, 0.0506829321, 0.44694671, 0.339641482, -0.0572569445, -0.559919596, -0.0473202169, 0.612989128, 0.634165406, 0.378141403, -0.455470681, -0.0332708657, -0.285203546, -0.52300024, 0.146062762, 0.143900007, -0.253096908, -0.122492813, 0.245238096, 0.256012172, -0.0255010668, -0.126703024, -0.158276811, -0.0148528507, 0.320309877, 0.261383206, 0.534014046, -0.137495875, 0.192852467, -0.118936479, -0.0230308473, -0.259963989, -0.140724778, 0.179532796, 0.611902237, 0.372040093, -0.260777652, -0.327730715, -0.0909247994, 0.410422176, 0.594913065, 0.630496025, -0.152438909, -0.57460463, -0.341402858, -0.397623032, -0.0528744012, -0.277876198, 0.20396173, -0.289548904, -0.140151143, 0.55270046, 0.290679365, 0.0602542721, 0.258478671, 0.193394065, 0.460692912, -0.138920575, 0.39920482, -0.334838927, 0.216209203, -0.264855325, -0.161031842, -0.268189907, 0.29284969, -0.236191094, -0.0166956261, 0.0339621268, -0.149809256, -0.0790201947, -0.0944195539, -0.144070089, -0.137076512, 0.168433636, 0.047758311, -0.276829809, -0.230432674, 0.050457269, 0.236678034, -0.0649672896, 0.211509973, -0.0608861297, 0.0291235447, -0.19902879, -0.180561647, -0.160639122, -0.038616091, 0.0980684757, -0.133503079, -0.0310977697, -0.247202516, 0.168405265, -0.028773427, 0.279736549, -0.0647393167, -0.0645705312, 0.134770274, 0.0459939539, -0.00396078825, -0.2287893, 0.0274106562, 0.137310475, 0.270051986, -0.117455378, -0.277544349, 0.247196347, -0.217389092, -0.0112026632, 0.0300299823, -0.0752307922, -0.222790837, 0.131495059, -0.131336629, 0.297023565, -0.217945933, 0.274777323, -0.16430147, 0.179341316, -0.148265958, 0.0911439657, -0.175390244, 0.0790438354, -0.123433307, 0.00217476487, 0.190110713, -0.0862111598, 0.0962934196, 0.161018938, 0.147482932, 0.00325238705, 0.0647659898, -0.130838737, 0.252144068, 0.269696951, -0.231494248, 0.27029565, 0.217938572, -0.0599677861, -0.170433387, 0.158861756, -0.034960635, 0.163598269, -0.128041163, 0.155549139, 0.2925044, -0.160537124, 0.249680787, -0.0774963722, -0.2721771, 0.019709859, -0.0353721678, 0.0361271054, 0.0226767361, -0.0563989282, -0.216894656, 0.0773308426, -0.0720873922, 0.240764648, -0.246120259, -0.216267735, 0.291011781, 0.2509453, 0.020124143, 0.452161998, 0.13976863, 0.655727446, 0.124746382, -0.128783569, -0.198993757, -0.316543877, 0.268099368, 0.482871532, 0.653967738, 0.668740809, -0.132674873, 0.0679067373, -0.0365645997, 0.593207955, 0.0921032429, -0.360375881, 0.334674001, -0.125949949, -0.303485006, 0.0778906569, -0.471386194, 0.293197244, -0.553772271, 0.407498211];
    bias_4 : ARRAY[0..31] OF REAL := [0, 0, 0.213209897, 0.00224766345, 0.172340766, -0.0173055902, 0.0912607461, 0.133293286, 0, 0, 0.180098847, -0.018521294, 0, 0.00024637449, 0.116646565, 0.071674265, 0.134868905, 0.19432874, -0.00654612528, 0.149317056, -0.0326505601, -0.0136953797, 0.252407193, -0.0200294089, 0.0553330183, -0.0194768831, 0.111973867, 0.0557610691, -0.00781303924, 0, -0.0180669241, 0.176333666];

    weights_6 : ARRAY[0..511] OF REAL := [-0.135647863, 0.0665159822, -0.0292185545, -0.333010912, 0.0224739611, 0.273968607, 0.0425424278, -0.20122692, 0.0297139585, -0.132199734, 0.312975675, 0.0767269731, 0.349180847, 0.0477670431, -0.176244125, 0.194731861, 0.333876282, 0.141886771, 0.336009353, -0.248086631, 0.0409471691, -0.306513041, 0.186116785, -0.0773225129, 0.291634947, 0.0548725724, 0.328215271, -0.311473459, 0.103085786, 0.170528144, 0.34468922, 0.0419202745, 0.394788474, 0.334831566, -0.306291282, -0.272091508, 0.31355834, -0.661192179, 0.612704575, 0.198251948, 0.0114442222, -0.656439364, 0.548780859, 0.536289871, 0.101797454, 0.124256417, 0.347800404, 0.635411799, 0.50685209, -0.416734278, 0.27322492, -0.191738039, -1.02211285, -0.183053732, 0.554450154, 0.880896509, 0.26146102, -0.0535854734, 0.718949437, -1.04767156, 0.749403, 1.11482191, -0.891946793, -0.15777126, 0.210133448, -0.509267807, -0.05602175, -0.985189438, 0.00128901307, -0.884256184, 0.483640701, 0.590210795, 0.0489467047, -1.15174282, 0.957749307, 0.412814796, 0.649967313, 0.314656258, -0.531283617, 0.895701468, 0.205082551, -0.104781367, -0.0700836107, -0.330424309, 0.20649974, 0.241561487, -0.138423324, -0.292210072, 0.249425754, -0.00774867041, -0.121094622, -0.214165822, 0.204258889, -0.068315506, 0.208929271, 0.0467472896, 0.0392961428, -0.255968034, 0.265627295, -0.255805552, 0.385933667, -0.74713403, 0.579089999, 0.228510171, 0.318567246, -0.520760357, 0.627676368, 0.270513475, 0.360449463, 0.0502105355, -0.364987731, 0.833422542, 0.527392805, -0.255664974, -0.28996411, -0.750532568, 0.421531379, -0.541681945, 0.582768142, 0.112681448, -0.110062517, -0.301942766, 0.530819297, 0.613372266, 0.542551696, 0.539943278, -0.442968607, 0.886211812, 0.0760379732, 0.0334706604, -0.302015215, -0.211100921, -0.223661095, -0.268729329, -0.00668153167, -0.300373912, 0.128985047, 0.320597857, -0.00192341208, 0.319881827, 0.113553643, 0.0549184382, 0.191299647, 0.0457511544, -0.236114904, 0.240684956, 0.0968763828, 0.201802462, 0.133858651, -0.0667561293, -0.349250197, 0.00946339965, -0.280319273, -0.205247894, 0.0616274476, 0.229204923, 0.18416968, 0.0436075032, 0.00413864851, -0.163686559, 0.636937678, 0.146068558, 0.325863332, -0.302803487, 0.470554948, -0.117045365, 0.285934895, 0.176876634, -0.243329793, -0.505519152, 0.657935739, 0.333084017, -0.129205912, 0.0559978262, -0.0628032461, 0.588446319, -0.201402411, 0.169912457, -0.341353059, 0.187180549, 0.268665344, 0.0983546376, -0.203235626, -0.260534525, 0.319570631, 0.0487997234, 0.183261901, 0.248321995, -0.320872784, -0.180871934, -0.127147004, -0.31985864, -0.112962991, 0.106948972, -0.328283668, -0.239465579, -0.262165189, 0.28056708, 0.326355428, 0.204828709, 0.139129937, -0.149088323, -0.110558346, 0.186144263, 0.0491915345, -0.350541413, 0.238233477, 0.0246281028, -0.1566028, -0.230589107, -0.0535046756, 0.0737761036, -0.254741699, 0.205023199, -0.315673649, 0.280965537, -0.293441355, 0.218738139, 0.367734969, -0.196078882, 0.370361924, 0.193879455, 0.0452488922, -0.114545994, -0.30581817, 0.5802176, -0.347579837, -0.139612094, -0.00964512862, -0.19519493, -0.0445733629, -0.226170242, 0.0519349612, -0.143849075, -0.272542179, -0.00320442836, -0.123143688, 0.01393383, 0.16650556, 0.312199682, 0.521462142, -0.698717296, 0.347500533, -0.0379418954, -1.06033659, -0.129335314, 0.697552145, 1.04649556, -0.293077409, -0.0837986544, 0.542610109, -0.738136351, 0.886999488, 0.948241889, -0.560702562, -0.0665787011, 0.0180195849, 0.558195949, -0.290952504, 0.0253968481, -0.163552955, 0.667888522, -0.442524314, -0.280109853, -0.173298553, 0.26672104, -0.238530472, -0.470692039, -0.562184513, -0.702730238, 0.802936792, -0.373625159, 0.532706141, 0.145392373, -0.205444589, -0.787096322, 0.642753303, -0.145530611, 0.391598552, -0.0361083113, 0.138522908, -0.372333139, 0.738909721, 0.0223644581, 0.416337907, 0.463038355, 0.0405754745, 0.47633335, 0.13967368, -0.232094303, 0.163171023, 0.200966477, 0.234083414, 0.222526982, -0.134308577, -0.0601005554, -0.204910815, -0.247846141, 0.155142844, -0.320930809, -0.106540993, -0.14928253, 0.177549616, -0.35453549, -0.529308617, 0.763332367, 0.250268638, 0.442752481, 0.189360455, 0.558145165, -0.134592041, -0.305548519, 0.193605855, 0.400314778, 0.0090786526, 0.207726285, -0.749656498, -0.515207767, 0.334976435, -0.198031411, -0.131912038, -0.131592691, 0.295713931, -0.110432744, 0.207850114, 0.228519902, -0.322944403, 0.205745518, 0.152548224, -0.258824557, -0.0689100325, 0.27036193, -0.281999707, 0.123070106, 0.155957073, 0.357466757, 0.0564233884, -0.147564873, 0.0125438273, -0.12932834, -0.278288633, 0.0384232178, 0.0997604877, -0.0953570604, 0.251122534, -0.0295221228, 0.169191852, 0.222821712, 0.127209648, -0.31985718, 0.183279127, -0.129776388, 0.21026434, 0.687215149, -0.0445205346, 0.319177359, 0.330201119, -0.184783027, 0.261288673, 0.0505578369, 0.0174904205, 0.26482895, 0.344652921, 0.421880275, -0.0841617584, -0.236179382, 0.232659146, 0.402864307, 0.706013203, -0.819276273, -0.163703024, 0.291181415, -0.409510285, 0.000160538417, 0.541411996, 0.686043322, -0.31384483, -0.127673626, 0.307931751, -0.605001032, 0.64253062, 0.438370287, -0.848982453, -0.240886152, 0.931743562, -0.965783894, -0.238229915, -0.157712385, -0.877239823, -0.095278956, 0.44741112, 0.853967726, -0.0178056527, -0.103886731, 0.80564028, -0.968454599, 0.721677959, 1.12857485, -0.925434291, -0.222055689, 0.23699683, -0.268652886, 0.101798773, -0.142202094, 0.145180136, 0.203968719, -0.153989911, -0.1920508, -0.298909485, -0.276199996, -0.0583957583, -0.219003186, 0.303088933, -0.223865673, 0.230530709, 0.132232457, 0.0104486933, 0.800574243, 0.0265724696, 0.15535742, 0.119418994, 0.672601938, -0.225837171, -0.324947923, -0.193773463, 0.62012434, -0.554603875, 0.255588531, -0.376292437, -0.421998858, 0.183003843, -0.271674037, -0.257813692, 0.797307849, 0.0660060197, 0.424774021, -0.127620295, 0.438901305, -0.284349501, -0.637869, 0.0118065793, 0.455551535, -0.198728397, -0.110163383, -0.460284293, -0.371639669, 0.594011843, -0.417290896, 0.201304272, 0.173167914, -0.042452842, 0.322171956, -0.115295038, 0.16096361, -0.082742922, -0.0433306694, 0.0841231719, 0.142255306, 0.169063866, -0.317796826, 0.132194802, -0.0199733973, -0.136090741, -0.155674621, 0.0232830942, 0.212380081, 0.230193347, 0.266435534, -0.244872332, -0.197124258, 0.162287802, -0.318706214, -0.139027536, 0.181346923, -0.205807194, 0.27788654, 0.0944553018, -0.0962616205, -0.287153482, 0.264811069, -0.285127491, 0.13410373, -0.329595774, -0.270726979, -0.0289029963, 0.103479207, -0.338335872, 0.323350459, -0.0978736579, 0.0324340165, 0.155721024, 0.0475811809, 0.319879353, -0.228012249, -0.212220758, -0.334938824, 0.653938711, -0.166639134, 0.0509224832, -0.606091082, 0.475326985, -0.658133268, 0.610506296, 0.0630735904, 0.0418764837, -0.740645945, 0.435194969, 0.345138729, 0.47352764, 0.261205703, 0.243571207, 0.732897043];
    bias_6 : ARRAY[0..15] OF REAL := [0.0584411658, 0.170095652, -0.0469134711, -0.0373878106, 0.16601558, 0.0378477573, 0.115304731, 0.0166916419, -0.014600764, 0.0359849781, 0.111261226, 0.119320944, -0.0391100943, 0.0337212235, 0.167460546, 0.134540975];

    weights_7 : ARRAY[0..47] OF REAL := [0.644716978, 0.081450209, -1.12863922, -0.968903542, 0.645160675, 0.41950199, 0.435314655, 0.385903418, -0.0415477604, -0.150881454, -1.18719673, 0.582273185, -0.0318484008, 0.768632352, -0.526957512, -0.30481708, -0.584626377, 0.566867292, 0.837831557, -0.107032165, -1.21557891, 1.23962617, -0.402116925, -0.195668131, 0.335846364, -0.2942307, -0.25329563, -0.284149855, -0.840044677, 1.02898753, 0.300938576, 0.188863322, -0.921342492, -0.490959615, 0.0181329921, -0.844524443, 1.08292305, -1.11623573, -0.29139027, 0.847201049, -0.69343847, 0.11735642, -1.05344462, 0.265259713, 0.63248992, 0.516839862, 0.564170122, -1.0380981];
    bias_7 : ARRAY[0..2] OF REAL := [-0.145640135, 0.0898162946, 0.0415015779];

END_VAR

VAR
    (* Merged variables from all regions *)
    buffer_0 : ARRAY[0..31] OF REAL;
    buffer_1 : ARRAY[0..31] OF REAL;

    (* Temporary computation variables *)
    i : DINT;
    j : DINT;
    t : DINT;
    sum : REAL;
    (* Computation helpers *)
    max_val : REAL;
    exp_val : REAL;
    exp_sum : REAL;
    (* Spatial loop variables *)
    oc : DINT;
    oh : DINT;
    ow : DINT;
    ic : DINT;
    kh : DINT;
    kw : DINT;
    ih : DINT;
    iw : DINT;
END_VAR

(* Forward pass execution *)

(* Region: r0 [ACYCLIC] *)
(* Acyclic Region r0 *)
(* Layer 0: Conv2D  in=1x1x1  out=32x1x1  kernel=1x1  stride=1x1  pad=(0, 0, 0, 0)  group=1 *)
FOR oc := 0 TO 31 DO
    FOR oh := 0 TO 0 DO
        FOR ow := 0 TO 0 DO
            sum := bias_0[oc];
            FOR ic := 0 TO 0 DO
                FOR kh := 0 TO 0 DO
                    FOR kw := 0 TO 0 DO
                        ih := oh * 1 - 0 + kh;
                        iw := ow * 1 - 0 + kw;
                        sum := sum + input_data * weights_0[oc * 1 + ic * 1 + kh * 1 + kw];
                    END_FOR;
                END_FOR;
            END_FOR;
            buffer_1[oc * 1 + oh * 1 + ow] := sum;
        END_FOR;
    END_FOR;
END_FOR;

(* Layer 1: Activation (RELU) *)
FOR i := 0 TO 31 DO
    buffer_0[i] := MAX(buffer_1[i], 0.0);
END_FOR;

(* Layer 2: Conv2D  in=32x1x1  out=32x1x1  kernel=1x1  stride=1x1  pad=(0, 0, 0, 0)  group=1 *)
FOR oc := 0 TO 31 DO
    FOR oh := 0 TO 0 DO
        FOR ow := 0 TO 0 DO
            sum := bias_2[oc];
            FOR ic := 0 TO 31 DO
                FOR kh := 0 TO 0 DO
                    FOR kw := 0 TO 0 DO
                        ih := oh * 1 - 0 + kh;
                        iw := ow * 1 - 0 + kw;
                        sum := sum + buffer_0[ic * 1 + ih * 1 + iw] * weights_2[oc * 32 + ic * 1 + kh * 1 + kw];
                    END_FOR;
                END_FOR;
            END_FOR;
            buffer_1[oc * 1 + oh * 1 + ow] := sum;
        END_FOR;
    END_FOR;
END_FOR;

(* Layer 3: Activation (RELU) *)
FOR i := 0 TO 31 DO
    buffer_0[i] := MAX(buffer_1[i], 0.0);
END_FOR;

(* Layer 4: Conv2D  in=32x1x1  out=32x1x1  kernel=1x1  stride=1x1  pad=(0, 0, 0, 0)  group=1 *)
FOR oc := 0 TO 31 DO
    FOR oh := 0 TO 0 DO
        FOR ow := 0 TO 0 DO
            sum := bias_4[oc];
            FOR ic := 0 TO 31 DO
                FOR kh := 0 TO 0 DO
                    FOR kw := 0 TO 0 DO
                        ih := oh * 1 - 0 + kh;
                        iw := ow * 1 - 0 + kw;
                        sum := sum + buffer_0[ic * 1 + ih * 1 + iw] * weights_4[oc * 32 + ic * 1 + kh * 1 + kw];
                    END_FOR;
                END_FOR;
            END_FOR;
            buffer_1[oc * 1 + oh * 1 + ow] := sum;
        END_FOR;
    END_FOR;
END_FOR;

(* Layer 5: Activation (RELU) *)
FOR i := 0 TO 31 DO
    buffer_0[i] := MAX(buffer_1[i], 0.0);
END_FOR;

(* Layer 6: Fused Linear + RELU *)
FOR j := 0 TO 15 DO
    sum := 0.0;
    FOR i := 0 TO 31 DO
        sum := sum + buffer_0[i] * weights_6[i * 16 + j];
    END_FOR;
buffer_1[j] := MAX(sum + bias_6[j], 0.0);
END_FOR;

(* Layer 7: Fused Linear + SOFTMAX *)
FOR j := 0 TO 2 DO
    sum := 0.0;
    FOR i := 0 TO 15 DO
        sum := sum + buffer_1[i] * weights_7[i * 3 + j];
    END_FOR;
output_data[j] := sum + bias_7[j];
END_FOR;

(* Softmax: find max *)
max_val := output_data[0];
FOR i := 1 TO 2 DO
    IF output_data[i] > max_val THEN
        max_val := output_data[i];
    END_IF;
END_FOR;

(* Softmax: compute exponentials and sum *)
exp_sum := 0.0;
FOR i := 0 TO 2 DO
    output_data[i] := EXP(output_data[i] - max_val);
    exp_sum := exp_sum + output_data[i];
END_FOR;

(* Softmax: normalize *)
FOR i := 0 TO 2 DO
    output_data[i] := output_data[i] / exp_sum;
END_FOR;

END_FUNCTION_BLOCK
